DATA_BLOCK "DB_AlarmLatch_Cylinder"
{ S7_Optimized_Access := 'TRUE' }
VERSION : 0.1
NON_RETAIN
"FB_AlarmLatch"
BEGIN
END_DATA_BLOCK
